// TwinCAT 3 PLC project Main_Control
// ProgramVersion: 3.1.4023.0
// libraries:
//   Tc2_Standard, * (Beckhoff Automation GmbH)
//   Tc2_System, * (Beckhoff Automation GmbH)
//   Tc3_Module, * (Beckhoff Automation GmbH)
// project tree:
//   DUTs/ E_EventType.TcDUT, Places_position.TcDUT, Positions.TcDUT, ST_Event.TcDUT
//   GVLs/ GVL.TcGVL
//   / PlcTask.TcTTO (not stored)
//   POUs/Heplcode/ EventLogger.TcPOU (not stored), FB_Time_Counter.TcPOU (not stored), F_UpdateEvent.TcPOU, INFO.TcPOU, Save_Error.TcPOU (not stored)
//   POUs/ MAIN.TcPOU
//   POUs/Motors/ Conveyor_1.TcPOU, Conveyor_2.TcPOU, Conveyor_3.TcPOU, Motor_Sorting.TcPOU
//   POUs/Positions/ Machine_Base_Position.TcPOU, Positions_init.TcPOU
// real-time tasks:
//   TASK PlcTask: cycle T#10ms, priority 20, ADS port 350
// I/O:
//   DEVICE Device 1 (EtherCAT) (disabled), AmsNetId 10.211.55.3.2.1
//     Term 1 (EK1200) [EK1200-7000 EtherCAT Power supply (1,5A E-Bus)]
//       Term 2 (EL1008) [EL1008 8Ch. Dig. Input 24V, 3ms]
//       Term 3 (EL1008) [EL1008 8Ch. Dig. Input 24V, 3ms]
//       Term 4 (EL1008) [EL1008 8Ch. Dig. Input 24V, 3ms]
//       Term 5 (EL3004) [EL3004 4Ch. Ana. Input +/-10V]
//       Term 6 (EL3004) [EL3004 4Ch. Ana. Input +/-10V]
//       Term 7 (EL9110) [EL9110 Power Supplier with LED (24V, Diagnostics)]
//       Term 8 (EL2008) [EL2008 8Ch. Dig. Output 24V, 0.5A]
//       Term 9 (EL2008) [EL2008 8Ch. Dig. Output 24V, 0.5A]
//       Term 10 (EL9110) [EL9110 Power Supplier with LED (24V, Diagnostics)]
//       Term 11 (EL2008) [EL2008 8Ch. Dig. Output 24V, 0.5A]
//       Term 12 (EL2008) [EL2008 8Ch. Dig. Output 24V, 0.5A]
//       Term 13 (EK1122) [EK1122 2 port EtherCAT junction]
//         Term 14 (EK1100) [EK1100 EtherCAT Coupler (2A E-Bus)]
//           Term 15 (EL1008) [EL1008 8Ch. Dig. Input 24V, 3ms]
//           Term 16 (EL1008) [EL1008 8Ch. Dig. Input 24V, 3ms]
//           Term 17 (EL9110) [EL9110 Power Supplier with LED (24V, Diagnostics)]
//           Term 18 (EL2008) [EL2008 8Ch. Dig. Output 24V, 0.5A]
//           Term 19 (EL2008) [EL2008 8Ch. Dig. Output 24V, 0.5A]
// variable links:
//   Main_Control/Main_Control Instance <-> Device 1 (EtherCAT)/Term 1 (EK1200)/Term 2 (EL1008)
//     PlcTask Inputs/MAIN.Inp_Part_at_Conveyor_1 <-> Channel 1/Input

// ---- DUTs/E_EventType.TcDUT
{attribute 'qualified_only'}
{attribute 'strict'}
TYPE E_EventType :
(
	Alarm := 0,
	Message:=1
);
END_TYPE

// ---- DUTs/Places_position.TcDUT
TYPE Places_position :
STRUCT
	Number				: INT;
	Coordinate_X_Axis	: INT;
	Coordinate_Y_Axis	: INT;
END_STRUCT
END_TYPE

// ---- DUTs/Positions.TcDUT
{attribute 'qualified_only'}
{attribute 'strict'}
TYPE Positions :
(
	Position_1 := 4100,
	Position_2 := 12300,
	Position_3 := 20500,
	Position_4 := 28700
);
END_TYPE

// ---- DUTs/ST_Event.TcDUT
TYPE ST_Event :
STRUCT
	What_happend			: STRING[20];
	sEventText				: STRING[255];
	eEventType				: E_EventType;
	eEventSeverity			: TcEventSeverity;
	dtTimeStamp				: DATE_AND_TIME;
END_STRUCT
END_TYPE

// ---- GVLs/GVL.TcGVL
{attribute 'qualified_only'}
VAR_GLOBAL
	M_Part_is_ready_for_sorting					: BOOL;
	M_Part_is_shipped_on_the_Conveyor_2			: BOOL;
	Part_is_Sorted								: BOOL;
END_VAR

VAR_GLOBAL PERSISTENT
	EventBuffer 								: ARRAY [1..500] OF ST_Event;
	Parts_Counter								: UINT:=0;
END_VAR

// ---- POUs/Heplcode/F_UpdateEvent.TcPOU
FUNCTION F_UpdateEvent
VAR_INPUT
	stEvent				: REFERENCE TO ST_Event;
END_VAR
VAR
	fbGETSYSTEMTIME 	: GETSYSTEMTIME;
	stFileTime 			: T_FILETIME;
END_VAR

fbGETSYSTEMTIME(timeLoDW=> stFileTime.dwLowDateTime, 
				timeHiDW=> stFileTime.dwHighDateTime);
stEvent.dtTimeStamp:= FILETIME_TO_DT(fileTime:=stFileTime);

END_FUNCTION

// ---- POUs/Heplcode/INFO.TcPOU
FUNCTION_BLOCK INFO
VAR_INPUT
END_VAR
VAR_OUTPUT
END_VAR
VAR
END_VAR

Couter_R_TRIG(
CLK:= , 
Q=> );

END_FUNCTION_BLOCK

// ---- POUs/MAIN.TcPOU
PROGRAM MAIN
VAR
	//Main Terminal INPUTS
		//Part 1(Conveyor 1)	
	Inp_Part_at_Conveyor_1								AT%I*: BOOL;
	Inp_Plunger_Parts_Container_In						AT%I*: BOOL;
	Inp_Plunger_Parts_Container_Out						AT%I*: BOOL;
	Inp_Part_On_Conveyor_1								AT%I*: BOOL;
	Inp_Part_in_front_of_Parts_Alignment				AT%I*: BOOL;
	Inp_Plunger_Parts_Alignment_Left_In					AT%I*: BOOL;
	Inp_Plunger_Parts_Alignment_Left_Out				AT%I*: BOOL;
	Inp_Plunger_Parts_Alignment_Right_In				AT%I*: BOOL;	
	
	Inp_Plunger_Parts_Alignment_Right_Out				AT%I*: BOOL;
	Inp_Plunger_Parts_Alignment_Above_In				AT%I*: BOOL;
	Inp_Plunger_Parts_Alignment_Above_Out				AT%I*: BOOL;
	Inp_Part_in_front_of_Crane							AT%I*: BOOL;
	Inp_Crane_In										AT%I*: BOOL;
	Inp_Crane_Out										AT%I*: BOOL;
	Inp_Crane_Above										AT%I*: BOOL;
	Inp_Crane_Below										AT%I*: BOOL;
	
	Inp_Motor_1_Protection_Switch_is_OK					AT%I*: BOOL;
	Inp_Base_Positions									AT%I*: BOOL;
	Inp_Start_Button									AT%I*: BOOL;
	Inp_Stop_Button										AT%I*: BOOL;
	
		//Part 2(Conveyor 2)	
	Inp_Conveyor_2_Palette_Left_Side					AT%I*: BOOL;
	Inp_Conveyor_2_Palette_Right_Side					AT%I*: BOOL;
	Inp_Palette_in_front_of_Tester						AT%I*: BOOL;
	Inp_Stopper_Below									AT%I*: BOOL;
	Inp_Stopper_Above									AT%I*: BOOL;
	Inp_Feedback_from_Tester							AT%I*: BOOL;
	Inp_Reserve_1										AT%I*: BOOL;
	Inp_Motor_2_Protection_Switch_is_OK					AT%I*: BOOL;
	
	Inp_Conveyor_2_Pallete_Slider_In					AT%I*: BOOL;
	Inp_Conveyor_2_Pallete_Slider_Out					AT%I*: BOOL;
	Inp_Feedback_from_Tester_GOOD_Part					AT%I*: BOOL;
	Inp_Feedback_from_Tester_BAD_Part					AT%I*: BOOL;
		
		//Part 3(Conveyor 3)
	Inp_Conveyor_3_Palette_Left_Side					AT%I*: BOOL;
	Inp_Conveyor_3_Palette_Right_Side					AT%I*: BOOL;	
	Inp_Conveyor_3_Pallete_Slider_In					AT%I*: BOOL;
	Inp_Conveyor_3_Pallete_Slider_Out					AT%I*: BOOL;	
	Inp_Motor_3_Protection_Switch_is_OK					AT%I*: BOOL;

	//Coupler	
		//Part 4(Sorting System)
	Inp_Sorter_in_Basik_Position						AT%I*: BOOL;
	Inp_Sorter_Plunger_Above							AT%I*: BOOL;
	Inp_Sorter_Plunger_Below							AT%I*: BOOL;
	Inp_Measuring_Bar_Sorting_Axis_X					AT%I*: INT;
	Inp_Measuring_Bar_Sorting_Axis_Y					AT%I*: INT;
	Inp_Form_is_Changed_Button							AT%I*: BOOL;
	

	//Main Terminal OUTPUTS
		//Part 1(Conveyor 1)	
	Out_Conveyor_1_Motor_On								AT%Q*: BOOL;
	Out_Plunger_Parts_Container_Drive_In				AT%Q*: BOOL;
	Out_Plunger_Parts_Container_Drive_Out				AT%Q*: BOOL;
	Out_Plunger_Parts_Alignment_Left_Drive_In			AT%Q*: BOOL;
	Out_Plunger_Parts_Alignment_Left_Drive_Out			AT%Q*: BOOL;
	Out_Plunger_Parts_Alignment_Right_Drive_In			AT%Q*: BOOL;		
	Out_Plunger_Parts_Alignment_Right_Drive_Out			AT%Q*: BOOL;
	Out_Plunger_Parts_Alignment_Above_Drive_In			AT%Q*: BOOL;
	
	Out_Plunger_Parts_Alignment_Above_Drive_Out			AT%Q*: BOOL;
	Out_Crane_Drive_In									AT%Q*: BOOL;
	Out_Crane_Drive_Out									AT%Q*: BOOL;
	Out_Crane_Drive_Up									AT%Q*: BOOL;
	Out_Crane_Drive_Down								AT%Q*: BOOL;
	
		//Part 2(Conveyor 2)	
	Out_Conveyor_2_Motor_On								AT%Q*: BOOL;
	Out_Stopper_Drive_Up								AT%Q*: BOOL;
	Out_Stopper_Drive_Down								AT%Q*: BOOL;
	Out_Conveyor_2_Pallete_Slider_Drive_In				AT%Q*: BOOL;
	Out_Conveyor_2_Pallete_Slider_Drive_Out				AT%Q*: BOOL;
	
		//Part 3(Conveyor 3)
	Out_Conveyor_3_Motor_On								AT%Q*: BOOL;	
	Out_Conveyor_3_Pallete_Slider_Drive_In				AT%Q*: BOOL;
	Out_Conveyor_3_Pallete_Slider_Drive_Out				AT%Q*: BOOL;

	//Coupler	
		//Part 4(Sorting System)
	Out_Sortierer_Pluger_Drive_Up						AT%Q*: BOOL;
	Out_Sortierer_Pluger_Drive_Down						AT%Q*: BOOL;	
	Out_Measuring_Bar_Sorting_Axis_X_Motor_On			AT%Q*: BOOL;
	Out_Measuring_Bar_Sorting_Axis_Y_Motor_On			AT%Q*: BOOL;
	Out_Sorter_Pluger_Pull_in							AT%Q*: BOOL;
	
	position:Positions;
	a:INT;
	motor_Sorting:Motor_Sorting;
	conveyor_1:Conveyor_1;
	conveyor_2:Conveyor_2;
	conveyor_3:Conveyor_3;
	Buffer_VAR_Feedback_from_Tester_GOOD_Part:BOOL;
	Buffer_VAR_Feedback_from_Tester_BAD_Part:BOOL;
	M_Machine_Release										: RS;
	Machine_Base_Position:Machine_Base_Position;
END_VAR

M_Machine_Release(
SET:= Inp_Start_Button AND Machine_Base_Position.BOOL_Base_Position, 
RESET1:= Inp_Stop_Button);

motor_Sorting(
	Inp_Conveyor_2_Palette_Right_Side_at_Sorter:= , 
	Inp_Sortierer_in_Basic_Position:= , 
	Inp_Sorter_Plunger_Above:= , 
	Inp_Sorter_Plunger_Below:= , 
	Inp_Measuring_Bar_Sorting_Axis_X:= , 
	Inp_Measuring_Bar_Sorting_Axis_Y:= , 
	Inp_Form_is_Changed_Button:= , 
	Out_Sorter_Pluger_Drive_Up=> , 
	BOOL_Feedback_from_Tester_GOOD_Part:= Buffer_VAR_Feedback_from_Tester_GOOD_Part, 
	BOOL_Feedback_from_Tester_BAD_Part:= Buffer_VAR_Feedback_from_Tester_BAD_Part, 
	Out_Sorter_Pluger_Drive_Down=> , 
	Out_Measuring_Bar_Sorting_Axis_X_Right_Rotation_Motor_On=> , 
	Out_Measuring_Bar_Sorting_Axis_Y_Right_Rotation_Motor_On=> , 
	Out_Measuring_Bar_Sorting_Axis_X_Left_Rotation_Motor_On=> , 
	Out_Measuring_Bar_Sorting_Axis_Y_Left_Rotation_Motor_On=> , 
	Out_Sorter_Pluger_Pull_in=> , 
	Palette_at_Sorter_is_free=> );
	
	conveyor_1(
	Inp_Part_at_Conveyor_1:= Inp_Part_at_Conveyor_1, 
	Inp_Plunger_Parts_Container_In:= Inp_Plunger_Parts_Container_In, 
	Inp_Plunger_Parts_Container_Out:= Inp_Plunger_Parts_Container_Out, 
	Inp_Part_On_Conveyor_1:= Inp_Part_On_Conveyor_1, 
	Inp_Part_in_front_of_Parts_Alignment:= Inp_Part_in_front_of_Parts_Alignment, 
	Inp_Plunger_Parts_Alignment_Left_In:= Inp_Plunger_Parts_Alignment_Left_In, 
	Inp_Plunger_Parts_Alignment_Left_Out:= Inp_Plunger_Parts_Alignment_Left_Out, 
	Inp_Plunger_Parts_Alignment_Right_In:= Inp_Plunger_Parts_Alignment_Right_In, 
	Inp_Plunger_Parts_Alignment_Right_Out:= Inp_Plunger_Parts_Alignment_Right_Out, 
	Inp_Plunger_Parts_Alignment_Above_In:= Inp_Plunger_Parts_Alignment_Above_In, 
	Inp_Plunger_Parts_Alignment_Above_Out:= Inp_Plunger_Parts_Alignment_Above_Out, 
	Inp_Part_in_front_of_Crane:= Inp_Part_in_front_of_Crane, 
	Inp_Crane_In:= Inp_Crane_In, 
	Inp_Crane_Out:= Inp_Crane_Out, 
	Inp_Crane_Above:= Inp_Crane_Above, 
	Inp_Crane_Below:= Inp_Crane_Below, 
	Inp_Motor_1_Protection_Switch_is_OK:= Inp_Motor_1_Protection_Switch_is_OK, 
	Inp_Base_Positions:= Inp_Base_Positions, 
	Out_Conveyor_1_Motor_On=> , 
	Out_Plunger_Parts_Container_Drive_In=> , 
	Out_Plunger_Parts_Container_Drive_Out=> , 
	Out_Plunger_Parts_Alignment_Left_Drive_In=> , 
	Out_Plunger_Parts_Alignment_Left_Drive_Out=> , 
	Out_Plunger_Parts_Alignment_Right_Drive_In=> , 
	Out_Plunger_Parts_Alignment_Right_Drive_Out=> , 
	Out_Plunger_Parts_Alignment_Above_Drive_In=> , 
	Out_Plunger_Parts_Alignment_Above_Drive_Out=> , 
	Out_Crane_Drive_In=> , 
	Out_Crane_Drive_Out=> , 
	Out_Crane_Drive_Up=> , 
	Out_Crane_Drive_Down=> , 
	Out_Crane_Take_a_Part=> , 
	M_Part_is_shipped_on_the_Conveyor_2=> );
	
	conveyor_2(
	Inp_Conveyor_2_Palette_Left_Side:= Inp_Conveyor_2_Palette_Left_Side, 
	Inp_Conveyor_2_Palette_Right_Side:= Inp_Conveyor_2_Palette_Right_Side, 
	Inp_Palette_in_front_of_Tester:= Inp_Palette_in_front_of_Tester, 
	Inp_Stopper_Below:= Inp_Stopper_Below, 
	Inp_Stopper_Above:= Inp_Stopper_Above, 
	BOOL_Feedback_from_Tester_GOOD_Part:= Buffer_VAR_Feedback_from_Tester_GOOD_Part, 
	BOOL_Feedback_from_Tester_BAD_Part:= Buffer_VAR_Feedback_from_Tester_BAD_Part, 
	Inp_Motor_2_Protection_Switch_is_OK:= Inp_Motor_2_Protection_Switch_is_OK, 
	Inp_Conveyor_2_Pallete_Slider_In:= Inp_Conveyor_2_Pallete_Slider_In, 
	Inp_Conveyor_2_Pallete_Slider_Out:= Inp_Conveyor_2_Pallete_Slider_Out, 
	Out_Conveyor_2_Motor_On=> , 
	Out_Stopper_Drive_Up=> , 
	Out_Stopper_Drive_Down=> , 
	Out_Conveyor_2_Pallete_Slider_Drive_In=> , 
	Out_Conveyor_2_Pallete_Slider_Drive_Out=> , 
	M_Conveyor_2_is_ready_to_take_Part_From_Conveyor_2=> , 
	M_Part_is_ready_for_Test=> );
	
	conveyor_3(
	Inp_Conveyor_3_Palette_Left_Side:= Inp_Conveyor_3_Palette_Left_Side, 
	Inp_Conveyor_3_Palette_Right_Side:= Inp_Conveyor_3_Palette_Right_Side, 
	Inp_Conveyor_3_Pallete_Slider_In:= Inp_Conveyor_3_Pallete_Slider_In, 
	Inp_Conveyor_3_Pallete_Slider_Out:= Inp_Conveyor_3_Pallete_Slider_Out, 
	Inp_Motor_3_Protection_Switch_is_OK:= Inp_Motor_3_Protection_Switch_is_OK, 
	Inp_Conveyor_2_Palette_Right_Side:= Inp_Conveyor_2_Palette_Right_Side, 
	Out_Conveyor_3_Motor_On=> , 
	Out_Conveyor_3_Pallete_Slider_Drive_In=> , 
	Out_Conveyor_3_Pallete_Slider_Drive_Out=> ,
	Out_Sortierer_Pluger_Drive_Up=> , 
	Out_Sortierer_Pluger_Drive_Down=> , 
	Out_Measuring_Bar_Sorting_Axis_X_Motor_On=> , 
	Out_Measuring_Bar_Sorting_Axis_Y_Motor_On=> , 
	Out_Sorter_Pluger_Pull_in=> );
	
	Machine_Base_Position(
	Inp_Base_Positions:= Inp_Base_Positions );
	
	IF Inp_Feedback_from_Tester_GOOD_Part OR Main.motor_Sorting.Write_BOOL_Feedback_from_Tester_GOOD_Part
		THEN Buffer_VAR_Feedback_from_Tester_GOOD_Part:=TRUE;
	END_IF
		IF Inp_Feedback_from_Tester_GOOD_Part=FALSE OR Main.motor_Sorting.Write_BOOL_Feedback_from_Tester_GOOD_Part=FALSE
		THEN Buffer_VAR_Feedback_from_Tester_GOOD_Part:=FALSE;
	END_IF
	
		IF Inp_Feedback_from_Tester_BAD_Part OR Main.motor_Sorting.Write_BOOL_Feedback_from_Tester_BAD_Part
		THEN Buffer_VAR_Feedback_from_Tester_BAD_Part:=TRUE;
	END_IF
		IF Inp_Feedback_from_Tester_BAD_Part=FALSE OR Main.motor_Sorting.Write_BOOL_Feedback_from_Tester_BAD_Part=FALSE
		THEN Buffer_VAR_Feedback_from_Tester_BAD_Part:=FALSE;
	END_IF

END_PROGRAM

// ---- POUs/Motors/Motor_Sorting.TcPOU
FUNCTION_BLOCK Motor_Sorting
VAR_INPUT
	Inp_Conveyor_2_Palette_Right_Side_at_Sorter						: BOOL;	
	Inp_Sortierer_in_Basic_Position									: BOOL;
	Inp_Sorter_Plunger_Above										: BOOL;
	Inp_Sorter_Plunger_Below										: BOOL;
	Inp_Measuring_Bar_Sorting_Axis_X								: INT;
	Inp_Measuring_Bar_Sorting_Axis_Y								: INT;
	Inp_Form_is_Changed_Button										: BOOL;
	BOOL_Feedback_from_Tester_GOOD_Part								: BOOL;
	BOOL_Feedback_from_Tester_BAD_Part								: BOOL;
END_VAR
VAR_OUTPUT
	Out_Sorter_Pluger_Drive_Up										: BOOL;	
	Out_Sorter_Pluger_Drive_Down									: BOOL;	
	Out_Measuring_Bar_Sorting_Axis_X_Right_Rotation_Motor_On		: BOOL;
	Out_Measuring_Bar_Sorting_Axis_Y_Right_Rotation_Motor_On		: BOOL;
	Out_Measuring_Bar_Sorting_Axis_X_Left_Rotation_Motor_On			: BOOL;
	Out_Measuring_Bar_Sorting_Axis_Y_Left_Rotation_Motor_On			: BOOL;
	Out_Sorter_Pluger_Pull_in										: BOOL;	
	Palette_at_Sorter_is_free										: BOOL;
	Write_BOOL_Feedback_from_Tester_GOOD_Part						: BOOL;
	Write_BOOL_Feedback_from_Tester_BAD_Part						: BOOL;
END_VAR
VAR
	positions_init													: Positions_init;
	Pluger_Below_TON_For_Drive										: TON;
	Pluger_Below_TON_For_Release									: TON;
	i																: INT := 1;
	Measuring_Bar_Sorting_Axis_X_Motor_Above_Sorting_Place			: BOOL;
	Measuring_Bar_Sorting_Axis_Y_Motor_Above_Sorting_Place			: BOOL;
	Measuring_Bar_Sorting_Axis_X_Motor_At_Start_Position			: BOOL;
	Measuring_Bar_Sorting_Axis_Y_Motor_At_Start_Position			: BOOL;
	Part_On_Place													: BOOL;
	Part_on_Palette_at_Sorter										: BOOL;
	Part_Is_taken													: BOOL;
	Form_for_parts_is_FULL											: BOOL;
	Couter_R_TRIG													: R_TRIG;
END_VAR

positions_init();

Pluger_Below_TON_For_Drive(IN:= Sorter_is_ready_for_sorting() AND Inp_Sorter_Plunger_Below, PT:= T#2S);


Pluger_Below_TON_For_Release(
	IN:= Measuring_Bar_Sorting_Axis_X_Motor_Above_Sorting_Place 
	AND Measuring_Bar_Sorting_Axis_Y_Motor_Above_Sorting_Place 
	AND Part_On_Place 
	AND Inp_Sorter_Plunger_Below, 
	PT:= T#2S);

//If Form is full
IF i<=9 
	THEN 
		Form_for_parts_is_FULL:=TRUE;
		i:=0;	
END_IF

IF Inp_Form_is_Changed_Button AND i<9 AND Main.M_Machine_Release.Q1
	THEN 
		Form_for_parts_is_FULL:=FALSE;
END_IF

IF BOOL_Feedback_from_Tester_BAD_Part AND Sorter_is_ready_for_sorting() AND Main.M_Machine_Release.Q1
	THEN 
		BAD_Part_Sorting();
END_IF

IF BOOL_Feedback_from_Tester_GOOD_Part AND Sorter_is_ready_for_sorting() AND Main.M_Machine_Release.Q1
	THEN 
		GOOD_Part_Sorting();
END_IF

ACTION BAD_Part_Sorting:
IF Inp_Measuring_Bar_Sorting_Axis_Y > positions_init.Current_Position[1].Coordinate_Y_Axis
	THEN 
		Out_Measuring_Bar_Sorting_Axis_Y_Left_Rotation_Motor_On:=TRUE;
END_IF
	
IF Inp_Measuring_Bar_Sorting_Axis_Y <= positions_init.Current_Position[1].Coordinate_Y_Axis
	THEN 
		Out_Measuring_Bar_Sorting_Axis_Y_Left_Rotation_Motor_On:=FALSE; 
		Measuring_Bar_Sorting_Axis_Y_Motor_Above_Sorting_Place:=TRUE;
END_IF
	
IF Inp_Measuring_Bar_Sorting_Axis_Y <= positions_init.Current_Position[1].Coordinate_Y_Axis AND Measuring_Bar_Sorting_Axis_Y_Motor_Above_Sorting_Place
	THEN
		Out_Sorter_Pluger_Pull_in:=FALSE;
		GVL.Part_is_Sorted:=TRUE;  
END_IF
	
IF Inp_Measuring_Bar_Sorting_Axis_Y <= positions_init.Current_Position[1].Coordinate_Y_Axis AND Measuring_Bar_Sorting_Axis_Y_Motor_Above_Sorting_Place
	AND GVL.Part_is_Sorted
	THEN 
		IF Inp_Measuring_Bar_Sorting_Axis_Y < positions_init.Current_Position[0].Coordinate_Y_Axis
			THEN 
				Out_Measuring_Bar_Sorting_Axis_Y_Right_Rotation_Motor_On:=TRUE;
		END_IF
	
		IF Inp_Measuring_Bar_Sorting_Axis_Y >= positions_init.Current_Position[0].Coordinate_Y_Axis
			THEN 
				Out_Measuring_Bar_Sorting_Axis_Y_Right_Rotation_Motor_On:=FALSE; 
				BOOL_Feedback_from_Tester_BAD_Part:=FALSE;								
				Couter_R_TRIG(CLK:= TRUE, Q=> );
		END_IF
END_IF	

IF 	Couter_R_TRIG.Q
	THEN
		GVL.Parts_Counter:=GVL.Parts_Counter+1;
END_IF
END_ACTION

ACTION GOOD_Part_Sorting:
//Step 1 : Plunger goes down for a Part
IF Sorter_is_ready_for_sorting() 
	AND GVL.M_Part_is_ready_for_sorting 
	AND Inp_Sorter_Plunger_Above 
	AND Part_on_Palette_at_Sorter 
	AND NOT Form_for_parts_is_FULL 
	THEN 
		Out_Sorter_Pluger_Drive_Up:=FALSE; 
		Out_Sorter_Pluger_Drive_Down:=TRUE;
		Part_On_Place:=FALSE;
END_IF

//Step 2 : Plunger takes a Part
IF Sorter_is_ready_for_sorting() AND Inp_Sorter_Plunger_Below
	THEN 
		Out_Sorter_Pluger_Pull_in:=TRUE; 
		Part_on_Palette_at_Sorter:=FALSE; 
		GVL.M_Part_is_ready_for_sorting	:=FALSE;
END_IF

//Step 3 : Plunger is waiting for a 2 Seconds and drives up
IF Sorter_is_ready_for_sorting() AND Pluger_Below_TON_For_Drive.Q
	THEN 
		Out_Sorter_Pluger_Drive_Down:=FALSE;
		Out_Sorter_Pluger_Drive_Up:=TRUE;
		Part_Is_taken:=TRUE;
END_IF

//Step 4 : Plunger goes to Parts place
IF Sorter_is_ready_for_sorting() AND Inp_Sorter_Plunger_Above AND Part_Is_taken
	THEN 
		Sorter_to_Parts_Place(); 
		Palette_at_Sorter_is_free:=TRUE;
END_IF

//Step 5 : Plunger puts Part to place
IF Measuring_Bar_Sorting_Axis_X_Motor_Above_Sorting_Place 
	AND Measuring_Bar_Sorting_Axis_Y_Motor_Above_Sorting_Place
	AND Inp_Sorter_Plunger_Above
	THEN 
		Out_Sorter_Pluger_Drive_Up:=FALSE;
		Out_Sorter_Pluger_Drive_Down:=TRUE;	
END_IF

//Step 6 : Plunger releases Part
IF Measuring_Bar_Sorting_Axis_X_Motor_Above_Sorting_Place 
	AND Measuring_Bar_Sorting_Axis_Y_Motor_Above_Sorting_Place 
	AND Inp_Sorter_Plunger_Below
	THEN 
		Out_Sorter_Pluger_Pull_in:=FALSE;
		Part_On_Place:=TRUE;
END_IF

//Step 7 : Plunger releases Part
IF Pluger_Below_TON_For_Release.Q
	THEN 
		Out_Sorter_Pluger_Drive_Down:=FALSE;
		Out_Sorter_Pluger_Drive_Up:=TRUE;
		Part_Is_taken:=FALSE;
END_IF

//Step 7 : Sorter goes to the start position
IF Measuring_Bar_Sorting_Axis_X_Motor_Above_Sorting_Place 
	AND Measuring_Bar_Sorting_Axis_Y_Motor_Above_Sorting_Place
	AND Inp_Sorter_Plunger_Above
 	AND Part_On_Place 
	AND Part_Is_taken=FALSE
		THEN 
			Sorter_to_Start();
			GVL.Part_is_Sorted:=TRUE;
			BOOL_Feedback_from_Tester_GOOD_Part:=FALSE; 
			Couter_R_TRIG(CLK:= TRUE, Q=> );
END_IF

IF 	Couter_R_TRIG.Q
	THEN
		GVL.Parts_Counter:=GVL.Parts_Counter+1;
END_IF
END_ACTION

METHOD PRIVATE Sorter_is_ready_for_sorting : BOOL
VAR_INPUT
END_VAR
IF 	Measuring_Bar_Sorting_Axis_X_Motor_At_Start_Position 
	AND Measuring_Bar_Sorting_Axis_Y_Motor_At_Start_Position
	AND Inp_Conveyor_2_Palette_Right_Side_at_Sorter
		THEN 
			Sorter_is_ready_for_sorting:=TRUE;
END_IF

IF 	Measuring_Bar_Sorting_Axis_X_Motor_At_Start_Position =FALSE 
	OR Measuring_Bar_Sorting_Axis_Y_Motor_At_Start_Position =FALSE
	OR Inp_Conveyor_2_Palette_Right_Side_at_Sorter  =FALSE
		THEN 
			Sorter_is_ready_for_sorting:=FALSE;
END_IF
END_METHOD

ACTION Sorter_to_Parts_Place:
FOR i :=1 TO 9 DO
	
	IF Inp_Measuring_Bar_Sorting_Axis_X < positions_init.Current_Position[i].Coordinate_X_Axis
		THEN 
			Out_Measuring_Bar_Sorting_Axis_X_Right_Rotation_Motor_On:=TRUE;
			Measuring_Bar_Sorting_Axis_X_Motor_Above_Sorting_Place:=FALSE; 
	END_IF
	
	IF Inp_Measuring_Bar_Sorting_Axis_X >= positions_init.Current_Position[i].Coordinate_X_Axis
		THEN 
			Out_Measuring_Bar_Sorting_Axis_X_Right_Rotation_Motor_On:=FALSE; 
			Measuring_Bar_Sorting_Axis_X_Motor_Above_Sorting_Place:=TRUE;
	END_IF
	
		IF Inp_Measuring_Bar_Sorting_Axis_Y < positions_init.Current_Position[i].Coordinate_Y_Axis
		THEN 
			Out_Measuring_Bar_Sorting_Axis_Y_Right_Rotation_Motor_On:=TRUE;
			Measuring_Bar_Sorting_Axis_Y_Motor_Above_Sorting_Place:=FALSE; 
	END_IF
	
	IF Inp_Measuring_Bar_Sorting_Axis_Y >= positions_init.Current_Position[i].Coordinate_Y_Axis
		THEN 
			Out_Measuring_Bar_Sorting_Axis_Y_Right_Rotation_Motor_On:=FALSE; 
			Measuring_Bar_Sorting_Axis_Y_Motor_Above_Sorting_Place:=TRUE;
	END_IF
	
END_FOR
END_ACTION

ACTION Sorter_to_Start:
IF Inp_Measuring_Bar_Sorting_Axis_X > positions_init.Current_Position[0].Coordinate_X_Axis
	THEN 
		Out_Measuring_Bar_Sorting_Axis_X_Left_Rotation_Motor_On:=TRUE; 
END_IF
	
IF Inp_Measuring_Bar_Sorting_Axis_X <= positions_init.Current_Position[0].Coordinate_X_Axis
	THEN 
		Out_Measuring_Bar_Sorting_Axis_X_Left_Rotation_Motor_On:=FALSE; 
		Measuring_Bar_Sorting_Axis_X_Motor_At_Start_Position:=TRUE;
END_IF
	
IF Inp_Measuring_Bar_Sorting_Axis_Y > positions_init.Current_Position[0].Coordinate_Y_Axis
	THEN 
		Out_Measuring_Bar_Sorting_Axis_Y_Left_Rotation_Motor_On:=TRUE;
END_IF
	
IF Inp_Measuring_Bar_Sorting_Axis_Y <= positions_init.Current_Position[0].Coordinate_Y_Axis
	THEN 
		Out_Measuring_Bar_Sorting_Axis_Y_Left_Rotation_Motor_On:=FALSE; 
		Measuring_Bar_Sorting_Axis_Y_Motor_At_Start_Position:=TRUE;
END_IF
END_ACTION

END_FUNCTION_BLOCK

// ---- POUs/Positions/Positions_init.TcPOU
FUNCTION_BLOCK Positions_init
VAR_INPUT
END_VAR
VAR_OUTPUT
END_VAR
VAR
	Current_Position: Array [0..10] of Places_position;
END_VAR

Current_Position[0].Number:=0;
Current_Position[0].Coordinate_X_Axis:=Positions.Position_1;
Current_Position[0].Coordinate_Y_Axis:=Positions.Position_2;

Current_Position[1].Number:=0;
Current_Position[1].Coordinate_X_Axis:=Positions.Position_1;
Current_Position[1].Coordinate_Y_Axis:=Positions.Position_2;

Current_Position[2].Number:=0;
Current_Position[2].Coordinate_X_Axis:=Positions.Position_1;
Current_Position[2].Coordinate_Y_Axis:=Positions.Position_2;

Current_Position[3].Number:=0;
Current_Position[3].Coordinate_X_Axis:=Positions.Position_1;
Current_Position[3].Coordinate_Y_Axis:=Positions.Position_2;

Current_Position[4].Number:=0;
Current_Position[4].Coordinate_X_Axis:=Positions.Position_1;
Current_Position[4].Coordinate_Y_Axis:=Positions.Position_2;

Current_Position[5].Number:=0;
Current_Position[5].Coordinate_X_Axis:=Positions.Position_1;
Current_Position[5].Coordinate_Y_Axis:=Positions.Position_2;

Current_Position[6].Number:=0;
Current_Position[6].Coordinate_X_Axis:=Positions.Position_1;
Current_Position[6].Coordinate_Y_Axis:=Positions.Position_2;

Current_Position[7].Number:=0;
Current_Position[7].Coordinate_X_Axis:=Positions.Position_1;
Current_Position[7].Coordinate_Y_Axis:=Positions.Position_2;

Current_Position[8].Number:=0;
Current_Position[8].Coordinate_X_Axis:=Positions.Position_1;
Current_Position[8].Coordinate_Y_Axis:=Positions.Position_2;

Current_Position[9].Number:=0;
Current_Position[9].Coordinate_X_Axis:=Positions.Position_1;
Current_Position[9].Coordinate_Y_Axis:=Positions.Position_2;

Current_Position[10].Number:=0;
Current_Position[10].Coordinate_X_Axis:=Positions.Position_1;
Current_Position[10].Coordinate_Y_Axis:=Positions.Position_2;

END_FUNCTION_BLOCK

// ---- POUs/Motors/Conveyor_1.TcPOU
FUNCTION_BLOCK Conveyor_1
VAR_INPUT
	Inp_Part_at_Conveyor_1									: BOOL;
	Inp_Plunger_Parts_Container_In							: BOOL;
	Inp_Plunger_Parts_Container_Out							: BOOL;
	Inp_Part_On_Conveyor_1									: BOOL;
	Inp_Part_in_front_of_Parts_Alignment					: BOOL;
	Inp_Plunger_Parts_Alignment_Left_In						: BOOL;
	Inp_Plunger_Parts_Alignment_Left_Out					: BOOL;
	Inp_Plunger_Parts_Alignment_Right_In					: BOOL;	
	
	Inp_Plunger_Parts_Alignment_Right_Out					: BOOL;
	Inp_Plunger_Parts_Alignment_Above_In					: BOOL;
	Inp_Plunger_Parts_Alignment_Above_Out					: BOOL;
	Inp_Part_in_front_of_Crane								: BOOL;
	Inp_Crane_In											: BOOL;
	Inp_Crane_Out											: BOOL;
	Inp_Crane_Above											: BOOL;
	Inp_Crane_Below											: BOOL;
	
	Inp_Motor_1_Protection_Switch_is_OK						: BOOL;
	Inp_Base_Positions										: BOOL;
END_VAR
VAR_OUTPUT
	Out_Conveyor_1_Motor_On									: BOOL;
	Out_Plunger_Parts_Container_Drive_In					: BOOL;
	Out_Plunger_Parts_Container_Drive_Out					: BOOL;
	Out_Plunger_Parts_Alignment_Left_Drive_In			  	: BOOL;
	Out_Plunger_Parts_Alignment_Left_Drive_Out				: BOOL;
	Out_Plunger_Parts_Alignment_Right_Drive_In			 	: BOOL;		
	Out_Plunger_Parts_Alignment_Right_Drive_Out				: BOOL;
	Out_Plunger_Parts_Alignment_Above_Drive_In				: BOOL;	
	Out_Plunger_Parts_Alignment_Above_Drive_Out				: BOOL;
	Out_Crane_Drive_In										: BOOL;
	Out_Crane_Drive_Out										: BOOL;
	Out_Crane_Drive_Up										: BOOL;
	Out_Crane_Drive_Down									: BOOL;
	Out_Crane_Take_a_Part									: BOOL;
	M_Part_is_shipped_on_the_Conveyor_2						: BOOL;
END_VAR
VAR
	TON_Plunger_Parts_Container_1Sec_open					: TON;
	M_Part_Loading											: BOOL;
	M_Conveyor_1_is_ready_to_ship_on_Conveyor_2				: BOOL;
END_VAR

TON_Plunger_Parts_Container_1Sec_open(IN:= Inp_Plunger_Parts_Container_In, PT:= T#1S, Q=> , ET=> );

IF 	Inp_Part_at_Conveyor_1 
	AND NOT Out_Conveyor_1_Motor_On 
	AND NOT Inp_Part_in_front_of_Crane 
	AND NOT Inp_Part_On_Conveyor_1	
	AND NOT Inp_Part_in_front_of_Parts_Alignment
	AND NOT M_Part_Loading
	AND Main.M_Machine_Release.Q1
	THEN
		Out_Plunger_Parts_Container_Drive_Out:=FALSE;
		Out_Plunger_Parts_Container_Drive_In:=TRUE;
END_IF

IF TON_Plunger_Parts_Container_1Sec_open.Q AND Main.M_Machine_Release.Q1
	THEN 
		Out_Plunger_Parts_Container_Drive_In:=FALSE;
		Out_Plunger_Parts_Container_Drive_Out:=TRUE;
END_IF

IF Inp_Part_On_Conveyor_1 AND Inp_Plunger_Parts_Container_Out AND Main.M_Machine_Release.Q1
	THEN 
		Out_Conveyor_1_Motor_On:=TRUE;
END_IF

IF Out_Conveyor_1_Motor_On AND Inp_Part_in_front_of_Parts_Alignment AND Main.M_Machine_Release.Q1
	THEN 
		Out_Plunger_Parts_Alignment_Left_Drive_In			  	 :=FALSE;
		Out_Plunger_Parts_Alignment_Right_Drive_In			 	 :=FALSE;
		Out_Plunger_Parts_Alignment_Above_Drive_In				 :=FALSE;
		Out_Plunger_Parts_Alignment_Left_Drive_Out				 :=TRUE;	
		Out_Plunger_Parts_Alignment_Right_Drive_Out				 :=TRUE;	
		Out_Plunger_Parts_Alignment_Above_Drive_Out				 :=TRUE;
END_IF

IF Inp_Part_in_front_of_Crane AND Inp_Crane_Above AND Main.M_Machine_Release.Q1
	THEN
		Out_Conveyor_1_Motor_On:=FALSE;
		Out_Plunger_Parts_Alignment_Left_Drive_Out				 :=FALSE;
		Out_Plunger_Parts_Alignment_Right_Drive_Out				 :=FALSE;
		Out_Plunger_Parts_Alignment_Above_Drive_Out				 :=FALSE;
		Out_Plunger_Parts_Alignment_Left_Drive_In			 	 :=TRUE;
		Out_Plunger_Parts_Alignment_Right_Drive_In			 	 :=TRUE;		
		Out_Plunger_Parts_Alignment_Above_Drive_In				 :=TRUE;	
		M_Conveyor_1_is_ready_to_ship_on_Conveyor_2				 :=TRUE;	
END_IF

IF M_Conveyor_1_is_ready_to_ship_on_Conveyor_2 AND Main.conveyor_2.M_Conveyor_2_is_ready_to_take_Part_From_Conveyor_2 AND Main.M_Machine_Release.Q1
	THEN
		Out_Crane_Drive_Up:=FALSE;
		Out_Crane_Drive_Down:=TRUE;
END_IF

IF Inp_Part_in_front_of_Crane AND Inp_Crane_Below AND Inp_Crane_In AND NOT Out_Crane_Take_a_Part AND Main.M_Machine_Release.Q1
	THEN 
		Out_Crane_Take_a_Part:=TRUE;
		M_Part_Loading:=TRUE;
END_IF	

IF Out_Crane_Take_a_Part AND Inp_Crane_Below AND Inp_Crane_In AND M_Part_Loading AND Main.M_Machine_Release.Q1
	THEN 
		Out_Crane_Drive_Down:=FALSE; 
		Out_Crane_Drive_Up:=TRUE;
END_IF

IF Out_Crane_Take_a_Part AND Inp_Crane_Above AND Inp_Crane_In AND M_Part_Loading AND Main.M_Machine_Release.Q1
	THEN 
		Out_Crane_Drive_In:=FALSE;
		Out_Crane_Drive_Out:=TRUE;
END_IF

IF Out_Crane_Take_a_Part AND Inp_Crane_Above AND Inp_Crane_Out AND M_Part_Loading AND Main.M_Machine_Release.Q1
	THEN 		
		Out_Crane_Drive_Up:=FALSE;
		Out_Crane_Drive_Down:=TRUE;
END_IF

IF Out_Crane_Take_a_Part AND Inp_Crane_Below AND Inp_Crane_Out AND M_Part_Loading AND Main.M_Machine_Release.Q1
	THEN	
		Out_Crane_Take_a_Part:=FALSE;
END_IF

IF NOT Out_Crane_Take_a_Part AND Inp_Crane_Below AND Inp_Crane_Out AND M_Part_Loading AND Main.M_Machine_Release.Q1
	THEN	
		Out_Crane_Drive_Down:=FALSE; 
		Out_Crane_Drive_Up:=TRUE;
END_IF

IF NOT Out_Crane_Take_a_Part AND Inp_Crane_Above AND Inp_Crane_Out AND Main.M_Machine_Release.Q1
	THEN	
		Out_Crane_Drive_Out:=FALSE;
		Out_Crane_Drive_In:=TRUE;
		M_Part_is_shipped_on_the_Conveyor_2:=TRUE;
		M_Conveyor_1_is_ready_to_ship_on_Conveyor_2:=FALSE;
		M_Part_Loading:=FALSE;
END_IF

END_FUNCTION_BLOCK

// ---- POUs/Motors/Conveyor_2.TcPOU
FUNCTION_BLOCK Conveyor_2
VAR_INPUT
	Inp_Conveyor_2_Palette_Left_Side						: BOOL;
	Inp_Conveyor_2_Palette_Right_Side						: BOOL;
	Inp_Palette_in_front_of_Tester							: BOOL;
	Inp_Stopper_Below										: BOOL;
	Inp_Stopper_Above										: BOOL;
	BOOL_Feedback_from_Tester_GOOD_Part						: BOOL;
	BOOL_Feedback_from_Tester_BAD_Part						: BOOL;
	Inp_Motor_2_Protection_Switch_is_OK						: BOOL;
	
	Inp_Conveyor_2_Pallete_Slider_In						: BOOL;
	Inp_Conveyor_2_Pallete_Slider_Out						: BOOL;
END_VAR
VAR_OUTPUT
	Out_Conveyor_2_Motor_On									: BOOL;
	Out_Stopper_Drive_Up									: BOOL;
	Out_Stopper_Drive_Down									: BOOL;
	Out_Conveyor_2_Pallete_Slider_Drive_In					: BOOL;
	Out_Conveyor_2_Pallete_Slider_Drive_Out					: BOOL;
	M_Conveyor_2_is_ready_to_take_Part_From_Conveyor_2		: BOOL;
	M_Part_is_ready_for_Test								: BOOL;
END_VAR
VAR
END_VAR

IF 	Inp_Conveyor_2_Palette_Left_Side AND Main.M_Machine_Release.Q1
	AND NOT Inp_Conveyor_2_Palette_Right_Side 
	AND NOT Inp_Palette_in_front_of_Tester 
	AND Inp_Stopper_Below 
	AND Inp_Conveyor_2_Pallete_Slider_In 
	AND NOT Out_Conveyor_2_Motor_On
	THEN
		M_Conveyor_2_is_ready_to_take_Part_From_Conveyor_2:=TRUE;
END_IF

IF 	NOT Inp_Conveyor_2_Palette_Left_Side AND Main.M_Machine_Release.Q1
	OR  Inp_Conveyor_2_Palette_Right_Side 
	OR Inp_Palette_in_front_of_Tester 
	OR NOT Inp_Stopper_Below 
	OR NOT Inp_Conveyor_2_Pallete_Slider_In 
	OR Out_Conveyor_2_Motor_On
	THEN 
		M_Conveyor_2_is_ready_to_take_Part_From_Conveyor_2:=FALSE;
END_IF

IF Main.conveyor_1.M_Part_is_shipped_on_the_Conveyor_2 AND NOT Inp_Conveyor_2_Palette_Right_Side AND Main.M_Machine_Release.Q1
	THEN  Out_Conveyor_2_Motor_On:=TRUE; GVL.M_Part_is_shipped_on_the_Conveyor_2:=FALSE;
END_IF

IF Inp_Palette_in_front_of_Tester AND Main.M_Machine_Release.Q1
	THEN  
		Out_Conveyor_2_Motor_On:=FALSE;
END_IF

IF Inp_Palette_in_front_of_Tester AND Out_Conveyor_2_Motor_On=FALSE AND Main.M_Machine_Release.Q1
	THEN 
		Out_Stopper_Drive_Down:=FALSE;
		Out_Stopper_Drive_Up:=TRUE;
END_IF

IF Inp_Stopper_Above AND NOT BOOL_Feedback_from_Tester_GOOD_Part AND NOT BOOL_Feedback_from_Tester_BAD_Part AND Main.M_Machine_Release.Q1
	THEN 
		M_Part_is_ready_for_Test:=TRUE;
END_IF

IF Inp_Stopper_Above AND (BOOL_Feedback_from_Tester_GOOD_Part OR BOOL_Feedback_from_Tester_BAD_Part) AND Main.M_Machine_Release.Q1
	THEN 
		Out_Stopper_Drive_Up:=FALSE; 
		Out_Stopper_Drive_Down:=TRUE; 
		M_Part_is_ready_for_Test:=FALSE;
END_IF

IF Inp_Stopper_Below AND (BOOL_Feedback_from_Tester_GOOD_Part OR BOOL_Feedback_from_Tester_BAD_Part) AND Main.M_Machine_Release.Q1
	THEN 
		Out_Conveyor_2_Motor_On:=TRUE;
END_IF

IF Inp_Conveyor_2_Palette_Right_Side AND (BOOL_Feedback_from_Tester_GOOD_Part OR BOOL_Feedback_from_Tester_BAD_Part) AND Main.M_Machine_Release.Q1
	THEN 
		Out_Conveyor_2_Motor_On:=FALSE;
		GVL.M_Part_is_ready_for_sorting:=TRUE;
END_IF

IF Main.conveyor_3.Out_Conveyor_3_Motor_On=FALSE AND Main.M_Machine_Release.Q1
	AND NOT Main.conveyor_3.Inp_Conveyor_3_Palette_Left_Side 
	AND NOT Main.conveyor_3.Inp_Conveyor_3_Palette_Right_Side
	AND Main.conveyor_3.Inp_Conveyor_3_Pallete_Slider_In
	AND GVL.Part_is_Sorted
	THEN 
		Out_Conveyor_2_Pallete_Slider_Drive_In:=FALSE;
		Out_Conveyor_2_Pallete_Slider_Drive_Out:=TRUE;
		GVL.Part_is_Sorted:=FALSE;
END_IF

IF Inp_Conveyor_2_Pallete_Slider_Out AND Main.M_Machine_Release.Q1
	THEN 
		Out_Conveyor_2_Pallete_Slider_Drive_Out:=FALSE; 
		Out_Conveyor_2_Pallete_Slider_Drive_In:=TRUE;
END_IF

END_FUNCTION_BLOCK

// ---- POUs/Motors/Conveyor_3.TcPOU
FUNCTION_BLOCK Conveyor_3
VAR_INPUT
	Inp_Conveyor_3_Palette_Left_Side					: BOOL;
	Inp_Conveyor_3_Palette_Right_Side					: BOOL;	
	Inp_Conveyor_3_Pallete_Slider_In					: BOOL;
	Inp_Conveyor_3_Pallete_Slider_Out					: BOOL;	
	Inp_Motor_3_Protection_Switch_is_OK					: BOOL;
	Inp_Conveyor_2_Palette_Right_Side					: BOOL;
END_VAR
VAR_OUTPUT
	Out_Conveyor_3_Motor_On								: BOOL;	
	Out_Conveyor_3_Pallete_Slider_Drive_In				: BOOL;
	Out_Conveyor_3_Pallete_Slider_Drive_Out				: BOOL;
	Out_Sortierer_Pluger_Drive_Up						: BOOL;
	Out_Sortierer_Pluger_Drive_Down						: BOOL;	
	Out_Measuring_Bar_Sorting_Axis_X_Motor_On			: BOOL;
	Out_Measuring_Bar_Sorting_Axis_Y_Motor_On			: BOOL;
	Out_Sorter_Pluger_Pull_in							: BOOL;
END_VAR
VAR
END_VAR

IF Inp_Conveyor_2_Palette_Right_Side AND Main.M_Machine_Release.Q1
	THEN 
		Out_Conveyor_3_Pallete_Slider_Drive_In:=FALSE; 
		Out_Conveyor_3_Pallete_Slider_Drive_Out:=TRUE;
END_IF
IF Inp_Conveyor_3_Pallete_Slider_Out AND Main.M_Machine_Release.Q1
	THEN 
		Out_Conveyor_3_Pallete_Slider_Drive_Out:=FALSE; 
		Out_Conveyor_3_Pallete_Slider_Drive_In:=TRUE;
END_IF

IF  Inp_Conveyor_3_Palette_Right_Side AND Main.M_Machine_Release.Q1
	AND NOT Inp_Conveyor_3_Palette_Left_Side 
	AND NOT Out_Conveyor_3_Motor_On
	THEN 
		Out_Conveyor_3_Motor_On:=TRUE;
END_IF

IF Inp_Conveyor_3_Palette_Left_Side AND Main.M_Machine_Release.Q1
	THEN 
		Out_Conveyor_3_Motor_On:=FALSE;
END_IF

END_FUNCTION_BLOCK

// ---- POUs/Positions/Machine_Base_Position.TcPOU
FUNCTION_BLOCK Machine_Base_Position
VAR_INPUT
	Inp_Base_Positions 									: BOOL;
END_VAR
VAR_OUTPUT
	Out_Conveyor_1_Motor_On								: BOOL;
	Out_Plunger_Parts_Container_Drive_In				: BOOL;
	Out_Plunger_Parts_Container_Drive_Out				: BOOL;
	Out_Plunger_Parts_Alignment_Left_Drive_In			: BOOL;
	Out_Plunger_Parts_Alignment_Left_Drive_Out			: BOOL;
	Out_Plunger_Parts_Alignment_Right_Drive_In			: BOOL;		
	Out_Plunger_Parts_Alignment_Right_Drive_Out			: BOOL;
	Out_Plunger_Parts_Alignment_Above_Drive_In			: BOOL;	
	Out_Plunger_Parts_Alignment_Above_Drive_Out			: BOOL;
	Out_Crane_Drive_In									: BOOL;
	Out_Crane_Drive_Out									: BOOL;
	Out_Crane_Drive_Up									: BOOL;
	Out_Crane_Drive_Down								: BOOL;
	
		//Part 2(Conveyor 2)	
	Out_Conveyor_2_Motor_On								: BOOL;
	Out_Stopper_Drive_Up								: BOOL;
	Out_Stopper_Drive_Down								: BOOL;
	Out_Conveyor_2_Pallete_Slider_Drive_In				: BOOL;
	Out_Conveyor_2_Pallete_Slider_Drive_Out				: BOOL;
	
		//Part 3(Conveyor 3)
	Out_Conveyor_3_Motor_On								: BOOL;	
	Out_Conveyor_3_Pallete_Slider_Drive_In				: BOOL;
	Out_Conveyor_3_Pallete_Slider_Drive_Out				: BOOL;
	Out_Sortierer_Pluger_Drive_Up						: BOOL;
	Out_Sortierer_Pluger_Drive_Down						: BOOL;	
	Out_Measuring_Bar_Sorting_Axis_X_Motor_On			: BOOL;
	Out_Measuring_Bar_Sorting_Axis_Y_Motor_On			: BOOL;
	Out_Sorter_Pluger_Pull_in							: BOOL;
	BOOL_Base_Position									: BOOL;
END_VAR
VAR
	TON_Incident_Protection								: TON;
END_VAR

TON_Incident_Protection(IN:= Inp_Base_Positions, PT:= T#3S, Q=> , ET=> );

//bring to Base Position 
IF Inp_Base_Positions AND TON_Incident_Protection.Q //goes after 3 seconds pushing
	THEN 
		//Conveyor 1	
	Out_Conveyor_1_Motor_On								:=FALSE;
	Out_Plunger_Parts_Container_Drive_In				:=FALSE;
	Out_Plunger_Parts_Alignment_Right_Drive_Out			:=FALSE;
	Out_Plunger_Parts_Alignment_Left_Drive_Out			:=FALSE;
	Out_Crane_Drive_Down								:=FALSE;	
	Out_Plunger_Parts_Alignment_Above_Drive_Out			:=FALSE;
	Out_Crane_Drive_Out									:=FALSE;
	Out_Crane_Drive_In									:=TRUE;
	Out_Plunger_Parts_Alignment_Above_Drive_In			:=TRUE;	
	Out_Plunger_Parts_Alignment_Right_Drive_In			:=TRUE;		
	Out_Crane_Drive_Up									:=TRUE;
	Out_Plunger_Parts_Container_Drive_Out				:=TRUE;
	Out_Plunger_Parts_Alignment_Left_Drive_In			:=TRUE;
	
		//Conveyor 2	
	Out_Conveyor_2_Motor_On								:=FALSE;
	Out_Stopper_Drive_Up								:=FALSE;
	Out_Conveyor_2_Pallete_Slider_Drive_Out				:=FALSE;
	Out_Stopper_Drive_Down								:=TRUE;
	Out_Conveyor_2_Pallete_Slider_Drive_In				:=TRUE;
	
		//Conveyor 3
	Out_Conveyor_3_Motor_On								:=FALSE;	
	Out_Sortierer_Pluger_Drive_Down						:=FALSE;	
	Out_Sorter_Pluger_Pull_in							:=FALSE;
	Out_Conveyor_3_Pallete_Slider_Drive_Out				:=FALSE;
	Out_Sortierer_Pluger_Drive_Up						:=TRUE;
	Out_Conveyor_3_Pallete_Slider_Drive_In				:=TRUE;

	Main.motor_Sorting.Sorter_to_Start();
END_IF

//check Base Position
IF 
			//Conveyor 1	
	Out_Conveyor_1_Motor_On									=FALSE
	AND Out_Plunger_Parts_Container_Drive_In				=FALSE
	AND Out_Plunger_Parts_Alignment_Right_Drive_Out			=FALSE
	AND Out_Plunger_Parts_Alignment_Left_Drive_Out			=FALSE
	AND Out_Crane_Drive_Down								=FALSE	
	AND Out_Plunger_Parts_Alignment_Above_Drive_Out			=FALSE
	AND Out_Crane_Drive_Out									=FALSE
	AND Out_Crane_Drive_In									=TRUE
	AND Out_Plunger_Parts_Alignment_Above_Drive_In			=TRUE	
	AND Out_Plunger_Parts_Alignment_Right_Drive_In			=TRUE		
	AND Out_Crane_Drive_Up									=TRUE
	AND Out_Plunger_Parts_Container_Drive_Out				=TRUE
	AND Out_Plunger_Parts_Alignment_Left_Drive_In			=TRUE
			//Conveyor 2	
	AND Out_Conveyor_2_Motor_On								=FALSE
	AND Out_Stopper_Drive_Up								=FALSE
	AND Out_Conveyor_2_Pallete_Slider_Drive_Out				=FALSE
	AND Out_Stopper_Drive_Down								=TRUE
	AND Out_Conveyor_2_Pallete_Slider_Drive_In				=TRUE
	
		//Conveyor 3
	AND Out_Conveyor_3_Motor_On								=FALSE	
	AND Out_Sortierer_Pluger_Drive_Down						=FALSE	
	AND Out_Sorter_Pluger_Pull_in							=FALSE
	AND Out_Conveyor_3_Pallete_Slider_Drive_Out				=FALSE
	AND Out_Sortierer_Pluger_Drive_Up						=TRUE
	AND Out_Conveyor_3_Pallete_Slider_Drive_In				=TRUE
	AND Main.motor_Sorting.Measuring_Bar_Sorting_Axis_X_Motor_Above_Sorting_Place
	AND Main.motor_Sorting.Measuring_Bar_Sorting_Axis_Y_Motor_Above_Sorting_Place
	
	THEN 
		BOOL_Base_Position:=TRUE;
	ELSE 
		BOOL_Base_Position:=FALSE;
END_IF

END_FUNCTION_BLOCK
